FUNCTION_BLOCK BeltLogic
VAR_INPUT
END_VAR
VAR_OUTPUT
END_VAR
VAR
	fallTrig: F_TRIG;
	fallTrigDetected: bool;
END_VAR

fallTrig(CLK:= gvl.FotocellOutput, Q => fallTrigDetected);

IF NOT LocalVariables.Locations[5].Item.Id = 0 THEN
	gvl.MotorBeltMove := TRUE;
ELSIF NOT gvl.FotocellOutput THEN
	gvl.MotorBeltMove := FALSE;
//ELSIF gvl.FotocellOutput THEN
//	LocalVariables.Locations[6].Item.Id := NULL;
//	LocalVariables.Locations[6].Item.Recipe := LocalVariables.Recipe;
END_IF

//IF fallTrigDetected THEN
//	LocalVariables.Locations[6].Item.Id := LocalVariables.Locations[5].Item.Id;
//	LocalVariables.Locations[6].Item.Recipe := LocalVariables.Locations[5].Item.Recipe;
//	LocalVariables.Locations[5].Item.Id := NULL;
//	LocalVariables.Locations[5].Item.Recipe := LocalVariables.Recipe;
//END_IF

END_FUNCTION_BLOCK

(* stored: Version 1.1.0.1, ProductVersion 3.1.4024.12
   POU BeltLogic: Id {f325210d-3b52-4054-8cf2-b1f617604848}, SpecialFunc None *)
